(* PLC project LD_FB.project, Inovance company InoProShop(V1.8.1.3) InoProShop(V1.8.1.3) *)
(* stored: creationDateTime 2025-03-12T13:02:00.3232061, modificationDateTime 2025-03-12T12:56:32.0628007 *)

CONFIGURATION Application
  RESOURCE Application ON PLC
    VAR_GLOBAL RETAIN PERSISTENT  (* GVL *)
      con1 : BOOL := TRUE;
      con2 : BOOL := TRUE;
      norm1 : INT;
    END_VAR
  END_RESOURCE
END_CONFIGURATION
